{attribute addProperty BoxType ""}
{attribute addProperty Id "_defaultSyncUnitTasks_97D7B59B216270DrivesSyncUnitTasks_97D7B59B216270"}
{attribute addProperty CRC "2991790823"}
{attribute addProperty SizeInBites "432"}
{attribute addProperty SizeInBytes "54"}
TYPE SyncUnits_B2531AE7 :
STRUCT
	{attribute addProperty Name "_default"}
	_default : SyncUnitTasks_97D7B59B;
	{attribute addProperty Name "Drives"}
	Drives : SyncUnitTasks_97D7B59B;
END_STRUCT
END_TYPE

(* stored: Version 1.2.0.0, ProductVersion 3.1.4024.9
   DUT SyncUnits_B2531AE7: Id {b3c259a0-8387-4066-be27-0dcaf75fa1fb} *)
